{attribute 'qualified_only'}
{attribute 'strict'}
TYPE E_Message_Temperature :
(
	eNoMessage := 0,
	eTooMuchTemperature := 1,
	eTemperatureConfigError := 2,
	eTemperatureGeneralError := 3,
	eTemperatureOverrangeError := 4,
	eTemperatureUnderrangeError := 5,
	eNoConnectionToBackend := 6
);
END_TYPE

(* stored: Version 1.1.0.1, ProductVersion 3.1.4024.6
   DUT E_Message_Temperature: Id {b1d72117-7d4a-4302-bddf-f6ccc0c14b98} *)
